TYPE TManagerPartStatus :
	(
		MPS_NoPart,
		MPS_NeedPearling,
		MPS_ReadyToMove,
		MPS_PartBusy
	);
END_TYPE

(* stored: Version 1.1.0.1, ProductVersion 3.1.4022.12
   DUT TManagerPartStatus: Id {b9cb790f-48cb-4d7b-90b5-b04263852bd5} *)
